TYPE ST_SequenceOptions :
STRUCT
	bSaveOnStopping:		BOOL;
END_STRUCT
END_TYPE

(* stored: Version 1.1.0.1
   DUT ST_SequenceOptions: Id {667cd9ec-fa82-0711-299f-39a01fc962f8} *)
